
// ===== library: MasterCopy "Copia de ESTRELLA -TRIANGULO" =====

FUNCTION_BLOCK "ESTRELLA -TRIANGULO"   // FB1, LAD
{ S7_Optimized_Access := 'FALSE' }
VERSION : 0.1
   VAR_INPUT
      MARCHA : Bool;
      PARO : Bool;
      TEMPORIZADOR : Timer;
      TIEMPO : S5Time;
   END_VAR
   VAR_OUTPUT
      LINEA : Bool;
      ESTRELLA : Bool;
      TRIANGULO : Bool;
   END_VAR
   VAR
      B0 : Bool;
      B1 : Bool;
      B2 : Bool;
      B3 : Bool;
      F4 : Bool;
      F5 : Bool;
      F6 : Bool;
      F7 : Bool;
   END_VAR
BEGIN

REGION Network 1
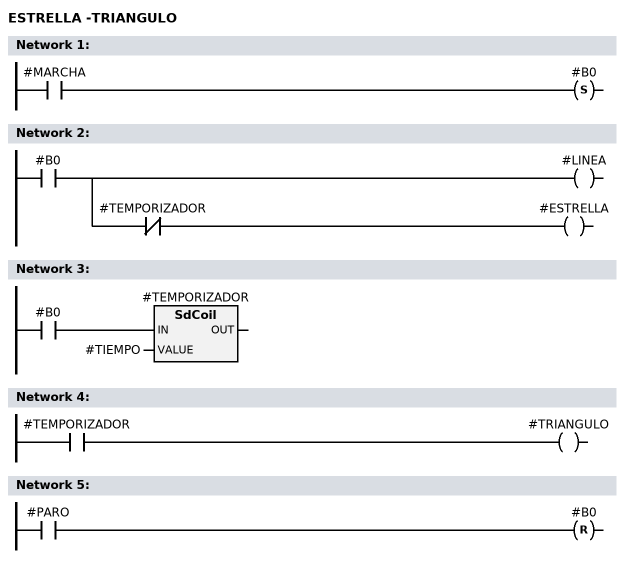
   RUNG wire#powerrail
      Contact( #MARCHA )
      S_Coil( #B0 )
   END_RUNG
   // the same network as SCL:
   IF #MARCHA THEN #B0 := TRUE; END_IF;
END_REGION

REGION Network 2
   RUNG wire#powerrail
      Contact( #B0 )
      wire#w1
      Coil( #LINEA )
   END_RUNG
   RUNG wire#w1
      I_Contact( #TEMPORIZADOR )
      Coil( #ESTRELLA )
   END_RUNG
   // the same network as SCL:
   #LINEA := #B0;
   #ESTRELLA := #B0 AND NOT #TEMPORIZADOR;
END_REGION

REGION Network 3
   // no SCL statement known for SdCoil: written as a call
   SdCoil(in := #B0, value := #TIEMPO, operand := #TEMPORIZADOR);
END_REGION

REGION Network 4
   RUNG wire#powerrail
      Contact( #TEMPORIZADOR )
      Coil( #TRIANGULO )
   END_RUNG
   // the same network as SCL:
   #TRIANGULO := #TEMPORIZADOR;
END_REGION

REGION Network 5
   RUNG wire#powerrail
      Contact( #PARO )
      R_Coil( #B0 )
   END_RUNG
   // the same network as SCL:
   IF #PARO THEN #B0 := FALSE; END_IF;
END_REGION
END_FUNCTION_BLOCK

// ===== library: MasterCopy "Copia de INTERMITENCIA" =====

FUNCTION_BLOCK "INTERMITENCIA"   // FB2, LAD
{ S7_Optimized_Access := 'FALSE' }
VERSION : 0.1
   VAR_INPUT
      "TIM 1" : S5Time;
      "TIM 2" : S5Time;
      TON : Timer;
      TOFF : Timer;
      MARCHA : Bool;
      PARO : Bool;
   END_VAR
   VAR_OUTPUT
      OUT : Bool;
   END_VAR
   VAR
      B0 : Bool;
      B1 : Bool;
      B2 : Bool;
      B3 : Bool;
   END_VAR
BEGIN

REGION Network 1
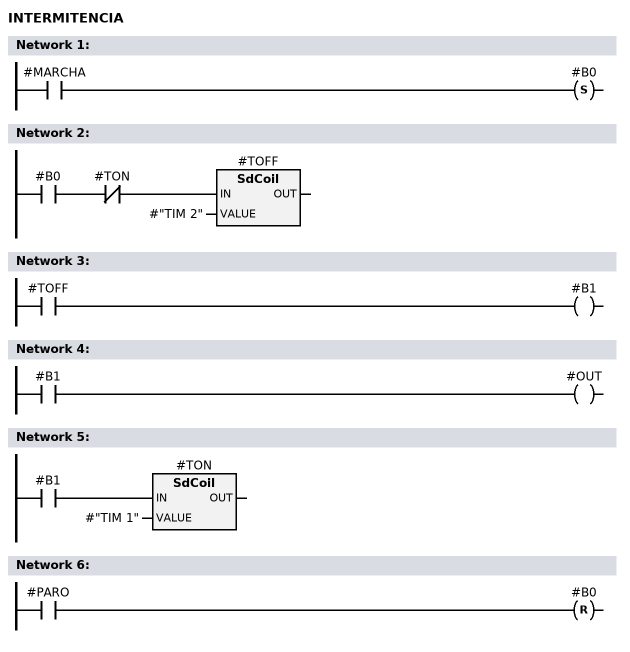
   RUNG wire#powerrail
      Contact( #MARCHA )
      S_Coil( #B0 )
   END_RUNG
   // the same network as SCL:
   IF #MARCHA THEN #B0 := TRUE; END_IF;
END_REGION

REGION Network 2
   // no SCL statement known for SdCoil: written as a call
   SdCoil(in := #B0 AND NOT #TON, value := #"TIM 2", operand := #TOFF);
END_REGION

REGION Network 3
   RUNG wire#powerrail
      Contact( #TOFF )
      Coil( #B1 )
   END_RUNG
   // the same network as SCL:
   #B1 := #TOFF;
END_REGION

REGION Network 4
   RUNG wire#powerrail
      Contact( #B1 )
      Coil( #OUT )
   END_RUNG
   // the same network as SCL:
   #OUT := #B1;
END_REGION

REGION Network 5
   // no SCL statement known for SdCoil: written as a call
   SdCoil(in := #B1, value := #"TIM 1", operand := #TON);
END_REGION

REGION Network 6
   RUNG wire#powerrail
      Contact( #PARO )
      R_Coil( #B0 )
   END_RUNG
   // the same network as SCL:
   IF #PARO THEN #B0 := FALSE; END_IF;
END_REGION
END_FUNCTION_BLOCK

// ===== library: MasterCopy "Copia de CONTADOR" =====

FUNCTION_BLOCK "CONTADOR"   // FB1, LAD
{ S7_Optimized_Access := 'FALSE' }
VERSION : 0.1
   VAR_INPUT
      UP : Bool;
      DOWN : Bool;
      RESET : Bool;
      PV : Real;
      DIGITO : Real;
   END_VAR
   VAR_OUTPUT
      OUT : Bool;
   END_VAR
   VAR
      B0 : Bool;
      B1 : Bool;
      B2 : Bool;
      CONTADOR : Real;
      CONTAJE : Real;
   END_VAR
   VAR_TEMP   // added for the SCL form of the ladder/FBD networks
      _w1 : Bool;
      _w2 : Bool;
   END_VAR
BEGIN

REGION Network 1
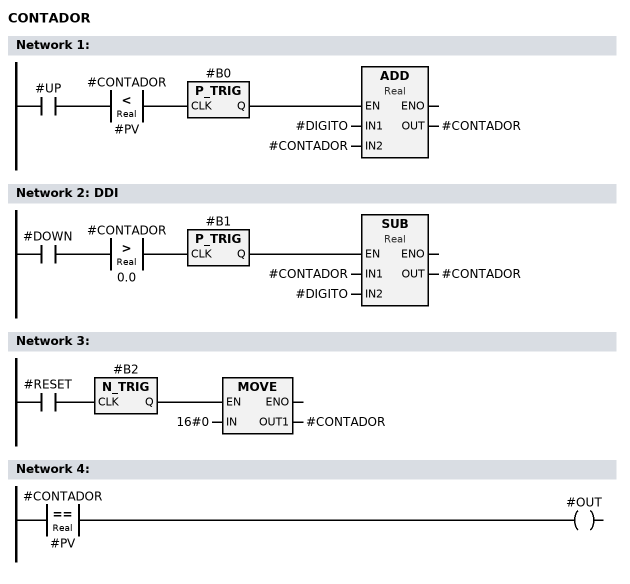
   RUNG wire#powerrail
      Contact( #UP )
      { S7_Templates := "SrcType := Real" } LT_Contact(in1 := #CONTADOR, in2 := #PV)
      P_Trig( #B0 )
      { S7_Templates := "SrcType := Real"; S7_GenerateENO := "TRUE" } Add(in1 := #DIGITO, in2 := #CONTADOR, out => #CONTADOR)
   END_RUNG
   // the same network as SCL:
   #_w1 := #UP AND (#CONTADOR < #PV);
   #_w2 := #_w1 AND NOT #B0;   // rising edge
   #B0 := #_w1;
   IF #_w2 THEN #CONTADOR := #DIGITO + #CONTADOR; END_IF;
END_REGION

REGION Network 2: DDI
   RUNG wire#powerrail
      Contact( #DOWN )
      { S7_Templates := "SrcType := Real" } GT_Contact(in1 := #CONTADOR, in2 := 0.0)
      P_Trig( #B1 )
      { S7_Templates := "SrcType := Real"; S7_GenerateENO := "TRUE" } Sub(in1 := #CONTADOR, in2 := #DIGITO, out => #CONTADOR)
   END_RUNG
   // the same network as SCL:
   #_w1 := #DOWN AND (#CONTADOR > 0.0);
   #_w2 := #_w1 AND NOT #B1;   // rising edge
   #B1 := #_w1;
   IF #_w2 THEN #CONTADOR := #CONTADOR - #DIGITO; END_IF;
END_REGION

REGION Network 3
   RUNG wire#powerrail
      Contact( #RESET )
      N_Trig( #B2 )
      { S7_GenerateENO := "TRUE" } Move(in := 16#0, out1 => #CONTADOR)
   END_RUNG
   // the same network as SCL:
   #_w1 := NOT #RESET AND #B2;   // falling edge
   #B2 := #RESET;
   IF #_w1 THEN #CONTADOR := 16#0; END_IF;
END_REGION

REGION Network 4
   RUNG wire#powerrail
      { S7_Templates := "SrcType := Real" } EQ_Contact(in1 := #CONTADOR, in2 := #PV)
      Coil( #OUT )
   END_RUNG
   // the same network as SCL:
   #OUT := #CONTADOR = #PV;
END_REGION
END_FUNCTION_BLOCK

// ===== library: MasterCopy "Copia de CONTADOR HORAS T Y PARCIAL" =====

FUNCTION_BLOCK "CONTADOR HORAS T Y PARCIAL"   // FB1, LAD
{ S7_Optimized_Access := 'FALSE' }
VERSION : 0.1
   VAR_INPUT
      MARCHA : Bool;
      PARO : Bool;
      "TIM 1" : Timer;
      "TIM 2" : Timer;
   END_VAR
   VAR_OUTPUT
      "SG.T" : Int;
      "MIN-T" : Int;
      "HORAS.T" : DInt;
      "SG.P" : Int;
      "MIN.P" : Int;
      "HORAS.P" : DInt;
   END_VAR
   VAR
      B0 : Bool;
      B1 : Bool;
      B2 : Bool;
      B3 : Bool;
      B4 : Bool;
      B5 : Bool;
      B6 : Bool;
      B7 : Bool;
      F10 : Bool;
      F11 : Bool;
      F12 : Bool;
      F13 : Bool;
      F14 : Bool;
      F15 : Bool;
      F16 : Bool;
      F17 : Bool;
      F20 : Bool;
      F21 : Bool;
      F22 : Bool;
      F23 : Bool;
      F24 : Bool;
      F25 : Bool;
   END_VAR
BEGIN
END_FUNCTION_BLOCK

// ===== library: MasterCopy "Copia de CALENDARIO" =====

FUNCTION_BLOCK "CALENDARIO"   // FB1, LAD
{ S7_Optimized_Access := 'FALSE' }
VERSION : 0.1
   VAR_INPUT
      CARGAR : Bool;
      "SG." : Int;
      "MIN." : Int;
      "HORAS." : Int;
      DIA : Int;
      MES : Int;
      AÑO : Int;
      "TIM 1" : Timer;
      "TIM 2" : Timer;
   END_VAR
   VAR_OUTPUT
      "SG 1" : Int;
      "MIN._1" : Int;
      "HORAS 1" : Int;
      DIA_1 : Int;
      MES_1 : Int;
      AÑO_1 : Int;
   END_VAR
   VAR
      B0 : Bool;
      B1 : Bool;
      B2 : Bool;
      B3 : Bool;
      B4 : Bool;
      B5 : Bool;
      B6 : Bool;
      B7 : Bool;
      F10 : Bool;
      F11 : Bool;
      F12 : Bool;
      F13 : Bool;
      F14 : Bool;
      F15 : Bool;
      F16 : Bool;
      F17 : Bool;
      F20 : Bool;
      F21 : Bool;
      F22 : Bool;
      F23 : Bool;
      F24 : Bool;
      F25 : Bool;
      F26 : Bool;
      F27 : Bool;
      "CSG." : Int;
      "CMIN." : Int;
      CHORAS : Int;
      CDIA : Int;
      CMES : Int;
      CAÑO : Int;
      DRESULTADO : Int;
      MRESULTADO : Int;
      RESULTADO : Int;
   END_VAR
BEGIN
END_FUNCTION_BLOCK